(* CODESYS project EAS_SCADA_BATCH.library
   Company: ESCARRE AUTOMATIZACION Y SERVICIOS sl
   Description: 1.1.3
      VAriable ALT fer IN_out
      1.1.2
      Incluir gestion PE
      1.1.1 
      Ajuste comunicacion ADS
      Ajuste tamaño constantes
   Version: 1.1.3
   Placeholder: EAS SCADA BATCH
   Author: EAS
   Title: EAS SCADA BATCH

Project tree, tasks and I/O mapping:
  libraries: Tc2_Standard, * (Beckhoff Automation GmbH); Tc2_System, * (Beckhoff Automation GmbH); Tc3_Module, * (Beckhoff Automation GmbH)
  DUTs/
    PE/
      ELEMENTS/
        data type E_Funcio
        data type PasCicle
        data type T_Compat
        data type T_funcio
        data type T_Sirena
      PE/
        data type PE
        data type PE_COM
      data type ATL
  GVLs/
    global variables Batch
    global variables CONSTANTS
  POUs/
    BATCH/
      function block CarregarFuncionsActivesAlDB [ST]
      function block ComprobarFuncionsPas [ST]
      function block Inic_Func_Actv [ST]
      function block Parar_Func_FiFuncio [ST]
      function block Parar_Func_Incomp [ST]
      function block PararTotesLesFuncions [ST]
      function block Salt [ST]
      function block SaltDePasEnUnCicle [ST]
    GestioPE/
      function block FunBck_v01 [ST]
      function block Func_Activa_v01 [ST]
    program pPE [ST]
  VISUs/
*)

// DUTs/PE/ELEMENTS/E_Funcio
TYPE E_Funcio :
STRUCT

	Cd_Funcio:WORD;
	Actv_Funcio:BOOL;
	ParamFunc:ARRAY [1..Max_ParamFunc] OF WORD;

END_STRUCT
END_TYPE

// DUTs/PE/ELEMENTS/PasCicle
TYPE PasCicle :
STRUCT
	Pas:WORD;
	Funcio:E_Funcio;

END_STRUCT
END_TYPE

// DUTs/PE/ELEMENTS/T_Compat
TYPE T_Compat :
STRUCT

	Funcio1:WORD;  			(*Codi de la primera funcio*)
	Funcio2:WORD;  			(*Codi de la segona funcio*)

END_STRUCT
END_TYPE

// DUTs/PE/ELEMENTS/T_funcio
TYPE T_funcio :
STRUCT

	Cd_funcio:WORD;												(*Codi de la funció*)
	DesFuncio:STRING(16);										(*Descripció de la funció*)
	Background:BOOL;												(*Indicació per si la funció es en backgraund o no*)
	FinFunc:ARRAY [1..max_FinFunc] OF WORD;					(*Funcions que s'han d'acabar al començar aquesta*)

END_STRUCT
END_TYPE

// DUTs/PE/ELEMENTS/T_Sirena
TYPE T_Sirena :
STRUCT
	Actv:BOOL;
	Rearme:BOOL;
END_STRUCT
END_TYPE

// DUTs/PE/PE/PE
TYPE PE :
STRUCT
	///1:manual  2: auto
	wAutoMan: WORD;
	xAuto: BOOL;
	xMan: BOOL;
	///Pas en Automatic, actual o ultim
	wStep: WORD;
	///Función fin de Ciclo
	wFEndCycle: WORD;
	///Tiempo Barcada
	wTBatch: WORD;
	///Tiempo Paso
	wTStep: WORD;
	///Tiempo mantenimiento
	wTMaint: WORD;
	xStartBatch: BOOL;
	xEndBatch: BOOL;
	///array alarmas
	axAlarm: ARRAY[1..Max_Alarmes] OF BOOL;
	///array Sirenas
	axHorn: ARRAY[1..Max_Alarmes] OF BOOL;
	///Pulsador Manual
	xPulMan: BOOL;
	///Pulsador Auto
	xPulAuto: BOOL;
END_STRUCT
END_TYPE

// DUTs/PE/PE/PE_COM
TYPE PE_COM :
STRUCT
	/// -------------------------------------------------------------------- 
	/// InfoBarcada 
	sBatch: STRING(10);
	diNum_Task: DWORD;
	sCdRecipe: STRING(24);
	sDesc_Recipe: STRING(50);
	sCdCycle: STRING(10);
	sDesc_Cycle: STRING(50);
	/// -------------------------------------------------------------------- 
	/// Ordenes PE 
	xToAutomatic: BOOL;
	xToManual: BOOL;
	xToStep: BOOL;
	xRunCycle: BOOL;
	xModifiedCycle: BOOL;
	xStopAlarm: BOOL;
	///Bit Para continuar programa
	xContProg: BOOL;
	///Bit indicacion al iniciar una añadida
	xStartTopping: BOOL;
	///Bit indicacion al finalizar una añadida
	xEndTopping: BOOL;
	///Bit indicacion para resetar los tiempos de la funcion al realizar un salto
	xResetStep: BOOL;
	xReset: BOOL;
	xResetFunc: BOOL;
	///word Per fer un canvi de Pas
	wNewStep: WORD;
	/// Pedir Dosificacion
	axDemandDos: ARRAY[1..max_tanks] OF BOOL;
	/// Numero Dosificacion 
	aiNumDos: ARRAY[1..max_tanks] OF WORD;
	/// OK Peticion Dosificacion
	axOkDemand: ARRAY[1..max_tanks] OF BOOL;
	/// OK  Dosificacion
	axOkDosage: ARRAY[1..max_tanks] OF BOOL;
	/// Tipo Dosificacion 1=Man 2=Auto 3=Mixta
	aiTypeDos: ARRAY[1..max_tanks] OF WORD;
	/// Dosificacion con Producto  Manual *
	axProdMan: ARRAY[1..max_tanks] OF BOOL;
	/// Error Dosificación  *
	axErrorDos: ARRAY[1..max_tanks] OF BOOL;
	/// Volumen dosificat
	aiVolumDos: ARRAY[1..max_tanks] OF DWORD;
	/// Tanque libre 
	axTankFree: ARRAY[1..max_tanks] OF BOOL;
	/// Prioridad
	aiPriority: ARRAY[1..max_tanks] OF WORD;
	/// Solo Disolver
	axOnlyDissol: ARRAY[1..max_tanks] OF BOOL;
END_STRUCT
END_TYPE

// DUTs/PE/ATL
TYPE ATL :
STRUCT
	///------OBLIGATORIO-------------------
	///Sistema PE Com
	PE_COM: PE_COM;
	///Sistema PE 
	PE: PE;
END_STRUCT
END_TYPE

// GVLs/Batch

VAR_GLOBAL RETAIN

(*=======================================	*)
(*					Estat del PE4							*)
(*=======================================	*)

(*Estat de PE4*)
	Func_Comp: ARRAY [1..Max_Compatibles] OF T_Compat;


(*=======================================	*)
(*			Variables de gestió de funcions				*)
(*=======================================	*)

(*Estat de lesFuncions *)
	Est_Func: ARRAY [1..Max_Funcions] OF E_Funcio;  		(*Estat actual de les funcions*)
	Est_F_PE4: ARRAY [1..Max_Funcions] OF E_Funcio;  		(*Estat de les funcions per les comunicacions del PE4*)
	Est_F_PE4_Ant: ARRAY [1..Max_Funcions] OF E_Funcio;  	(*Estat de les funcions per les comunicacions del PE4*)


(* *)
	Config_Func: ARRAY  [1..Max_Funcions] OF t_funcio;		(*Configuració de les funcios *)
	Func_Actives: ARRAY [1..Max_Func_Pas] OF WORD;		(* DB que indica en automaatic les funcions que estan en marcha en automatic*)


(*=======================================	*)
(*			Variables de gestió de cicle					*)
(*=======================================	*)

(*Cicles*)
	Cicle0: ARRAY [1..max_PasCicle] OF PasCicle;  			(*Cicle Actual de treball*)
	CicleRebut: ARRAY [1..max_PasCicle] OF PasCicle;  		(*Cicle Rebut*)


	

(*=======================================	*)
(*			Botons Auto/Man								*)
(*=======================================	*)

	PulsadorManual:BOOL;
	PulsadorAutomatic:BOOL;

(*=======================================	*)
(*			Marcas Internes								*)
(*=======================================	*)

	InicioCiclo:BOOL;


END_VAR


VAR_GLOBAL

(*=======================================	*)
(*			Maquina paralel 								*)
(*=======================================	*)

	TipoParalelo:WORD;
	MaquinaEnParalel:BOOL:=FALSE;
	Master:BOOL;
	Slave:BOOL;
	Pas_M:DWORD;
	Pas_S1:DWORD;
	Pas_S2:DWORD;
	Pas_S3:DWORD;
	Pas_S4:DWORD;
	Tipus_P:DWORD;
	Preparat_C_local:BOOL;
	He_C_local:BOOL;
	Ordre_C:BOOL;
	Ordre_C_Master:BOOL;
	Preparat_C_S1:BOOL;
	Preparat_C_S2:BOOL;
	Preparat_C_S3:BOOL;
	Preparat_C_S4:BOOL;
	He_C_S1:BOOL;
	He_C_S2:BOOL;
	He_C_S3:BOOL;
	He_C_S4:BOOL;
	Fi_C:BOOL;
	Fi_C_master:BOOL;



(*			CONSERVAR  COMPATIBILITAT				*)

	EsperaParalelPerSaltar:BOOL;
	SaltdePas:BOOL;


END_VAR

// GVLs/CONSTANTS

VAR_GLOBAL CONSTANT

(*=======================================	*)
(*			Carregar Constants						*)
(*=======================================	*)
	Max_Funcions:WORD:=128;
	Max_ParamFunc:WORD:=9;
	max_FinFunc:WORD:=5;
	max_PasCicle:WORD:=256;
	Max_Compatibles:WORD:=32;
	Max_Func_Pas:WORD:=12;
	Max_Tanks:WORD:=4;
	Max_Alarmes:WORD:=128;

END_VAR


(*********************************************************************


	Max_ParamFixes:WORD:=150;
	Max_DBFiFuncio: WORD:=640 ;				(* Es calcula com    (Max_Funcions*Max_FinFunc)   *)
	Max_ElementsCicle: WORD:=2816 ;		(* Es calcula com    (Max_PasCicle*(Max_ParamFunc+2))  *)
	Max_DBIncompatibles: WORD:=128;			(* Es calcula com    (Max_Compatibles*2)  *)
	Max_Inputs: WORD:=128;
	Max_Outputs: WORD:=128;
	Max_Analog: WORD:=128;
	Num_Prod_Dos:WORD:=10;         					(* Numero maximo de productos en una dosificación*)
	Max_Prod_Dos:WORD:=128;							(* Productos en una dosificadora*)
	Max_Valv_Dos:WORD:=128;							(* Valvulas en una dosificadora*)
	Max_Alarmes:WORD:=128;



***************************************************************************)

// POUs/BATCH/CarregarFuncionsActivesAlDB
FUNCTION_BLOCK CarregarFuncionsActivesAlDB

(***********************************************************************
Aquest Bloc Carrega les Funcions actives al "DB d'estat de les funcions"
al "DB de funcions actives".   
************************************************************************)

VAR_INPUT
	EstatFuncions: ARRAY [1..max_funcions] OF E_Funcio;
END_VAR

VAR_OUTPUT
	FuncionsActives:ARRAY [1..Max_Func_Pas] OF WORD;
END_VAR

VAR
	Punter:WORD;
	PunterDB:WORD;
	inicialitzaDB: Inic_Func_Actv;
	DB_ple: BOOL;

END_VAR

inicialitzaDB(Func_Actv:= FuncionsActives);
DB_Ple:=FALSE;
punter:=1;
punterDB:=1;
WHILE (punter<=max_funcions)AND NOT(DB_Ple)
	DO
		IF EstatFuncions[punter].Actv_Funcio
			THEN
				FuncionsActives[PunterDB]:=EstatFuncions[punter].Cd_Funcio;
				PunterDB:=PunterDB+1;
				IF punterDB>Max_Func_Pas
					THEN
						DB_ple:=TRUE;
				END_IF
		END_IF
		punter:=punter+1;
END_WHILE

END_FUNCTION_BLOCK

// POUs/BATCH/Inic_Func_Actv
FUNCTION_BLOCK Inic_Func_Actv

(*********************************************************
Reinicia el DB de les funcions actives
***********************************************************)

VAR_IN_OUT
	Func_Actv: ARRAY [1..Max_Func_Pas] OF WORD;		(* DB que indica en automaatic les funcions que estan en marcha en automatic*)
END_VAR

VAR
	Punter: WORD;
END_VAR

Punter:=1;

REPEAT
	Func_Actv[punter]:=0;
	Punter:=Punter+1;
UNTIL
	Punter>Max_Func_Pas
END_REPEAT

END_FUNCTION_BLOCK

// POUs/BATCH/ComprobarFuncionsPas
FUNCTION_BLOCK ComprobarFuncionsPas

(************************************************************
Aquest Bloc Comproba les funcions actves que hi ha en aquest
pas i quan acaben dona l'ordr de canviar de pas.
**************************************************************)

VAR_INPUT
	Estat_F: ARRAY [1..Max_Funcions] OF E_Funcio;
	Tipus_F:ARRAY [1..Max_Funcions] OF T_Funcio;
	FuncionsActives:ARRAY [1..Max_Func_Pas] OF WORD;
END_VAR

VAR_OUTPUT
	AumentaPas:BOOL;
END_VAR

VAR
	Punter: WORD;
	Aumenta: BOOL;
	TempoPAS:TON;

END_VAR

(*Inicialitzar els punters*)
Punter:=1;
Aumenta:=TRUE;

REPEAT
	IF (FuncionsActives[Punter]<>0)AND((Estat_F[FuncionsActives[Punter]].Actv_Funcio=TRUE)AND(Tipus_F[FuncionsActives[Punter]].Background=FALSE))
		THEN
			Aumenta:=FALSE;
	END_IF
	Punter:=Punter+1;
UNTIL
	(Punter>Max_Func_Pas)OR(Aumenta=FALSE)
END_REPEAT

TempoPAS
	(IN:=Aumenta ,
	PT:=t#500ms ,
	Q=>AumentaPas ,
	ET=> );

END_FUNCTION_BLOCK

// POUs/BATCH/Parar_Func_FiFuncio
FUNCTION_BLOCK Parar_Func_FiFuncio

(**************************************************
Para les funcions del "DB de l'estat de funcions" 
depenen de la funcio de la entreda per "fifuncion"
***************************************************)

VAR_INPUT
	Tipus_Funcio:T_funcio;
END_VAR
VAR_OUTPUT
END_VAR
VAR_IN_OUT
	Estat_F: ARRAY [1..Max_Funcions] OF E_Funcio;
END_VAR
VAR
	PunterFiFunc:WORD;
	FuncioIncompat: WORD;
END_VAR

(*..................	Parar les funcions per fin función..................................	*)
PunterFiFunc:=1;
WHILE (PunterFiFunc <= max_FinFunc) DO
	FuncioIncompat :=Tipus_funcio.FinFunc[PunterFiFunc];
	IF FuncioIncompat <>0
		THEN
			Estat_F [FuncioIncompat].Actv_Funcio:=FALSE;
	END_IF
	PunterFiFunc:=PunterFiFunc+1;
END_WHILE

END_FUNCTION_BLOCK

// POUs/BATCH/Parar_Func_Incomp
FUNCTION_BLOCK Parar_Func_Incomp
(************************************************************
L'hi introduim una funció i el el bloc para les funcions del 
"DB estat de les funcions" depenen del 
"DB de compatibilitat"
**************************************************************)
VAR_INPUT
	Funcio:WORD;  (*Funcio que s'ha de parar*)
END_VAR

VAR_OUTPUT
END_VAR

VAR_IN_OUT
	DB_Comp:ARRAY [1..Max_Compatibles] OF T_Compat;
	Estat_F: ARRAY [1..Max_Funcions] OF E_Funcio;
END_VAR

VAR
	PunterEstat:WORD;
	PunterComp:WORD;
END_VAR

(*Mirar si hi ha alguna funció incompatible amb la nova funció*)
PunterEstat:=1;
PunterComp:=1;
REPEAT
	IF DB_Comp[PunterComp].Funcio1=Funcio
		THEN
			PunterEstat:=DB_Comp[PunterComp].Funcio2;
			Estat_F[PunterEstat].Actv_Funcio:=FALSE;
	END_IF
	PunterComp:=PunterComp+1;
UNTIL
	(PunterComp>Max_Compatibles)
END_REPEAT

END_FUNCTION_BLOCK

// POUs/BATCH/PararTotesLesFuncions
FUNCTION_BLOCK PararTotesLesFuncions
(********************************************************
Parar totes les funcions del "DB estat"
*********************************************************)
VAR_IN_OUT
	Estat_F: ARRAY [1..Max_Funcions] OF E_Funcio;
END_VAR

VAR
	Punter: WORD;
END_VAR

(*Inicialitzar els punters*)
Punter:=1;


WHILE (Punter <= Max_Funcions) DO
	IF Estat_F[Punter].Actv_Funcio=TRUE
		THEN
			Estat_F [Punter].Actv_Funcio:=FALSE;
	END_IF
	Punter:=Punter+1;
END_WHILE

END_FUNCTION_BLOCK

// POUs/BATCH/Salt
FUNCTION_BLOCK Salt
(************************************************************
Salta del "Pas inicial" al "Pas Final"  del  "BDCicle"
**************************************************************)
VAR_INPUT
	PasInicial:DWORD;
	PasFinal:DWORD;
END_VAR

VAR_IN_OUT


END_VAR

VAR

	FIFuncio:Parar_Func_FiFuncio;
	Incompatibles:Parar_Func_Incomp;
	PunterCicle:WORD;					(* Aquest valor marca la popsició del db de cicle on estem independent del pas de cicle *)
	T_Func_Act:T_Funcio;				(* Funcio que indica el punterCicle *)

	codi: WORD;

	Est_Func_0: ARRAY [1..Max_Funcions] OF E_Funcio;  		(*Estat de les funcions a cero per reiniciar l'estat*)
END_VAR

(*,,,,,,,,,,,,,,,,,,,,Carregar la posició inicial depenen si es salta desde:
				el pas cero: carerega d'un cicle nou
				un pas en concret: salt sobre el cicle que ja està carregat ,,,,,,,,,,,,,,,,,,,,,  *)

IF PasInicial=0
	THEN
		(*Posar Punter al primer pas*)
		PunterCicle:=1;
		(*Inicialitzar el estat de les funcions*)
		Est_Func:=Est_Func_0;
	ELSE
		(*Buscar Punter Cicle del pas inicial*)
		PunterCicle:=0;
		REPEAT
			PunterCicle := PunterCicle+1;
		UNTIL
			(((Cicle0[PunterCicle].Pas=PasInicial)AND(Cicle0[PunterCicle+1].Pas<>PasInicial)) OR (PunterCicle>=max_PasCicle))
		END_REPEAT
		PunterCicle := PunterCicle+1;      (*02/06/05*)
END_IF

(*,,,,,,,,,,,,,,,,,,,,Bucle de control,,,,,,,,,,,,,,,,,,,,,,,,,,,,,,,,,,,,,,,,,,,,,,,,,,,,,,,,,,,,,	*)

REPEAT
(*.................. Carregar la funció del pas............................................. *)
		codi:=Cicle0[PunterCicle].Funcio.Cd_Funcio;
		IF codi<>0 THEN
		T_Func_Act:=Config_Func[codi];
		END_IF
(*..................	Parar les funcions incompatibles..................................	*)
		Incompatibles(
			Funcio:=T_Func_Act.Cd_funcio ,
			DB_Comp:= Func_Comp ,
			Estat_F:= Est_Func );

(*..................	Activar si es en Background ........................................	*)
		IF T_Func_Act.Background=TRUE
			THEN
				Est_Func[T_Func_Act.Cd_Funcio] := Cicle0[PunterCicle].Funcio ; 	(*Carregar parametres*)
				Est_Func[T_Func_Act.Cd_Funcio].Actv_Funcio:=TRUE;			(*Posar la funció en actiu*)
		END_IF

(*..................	Parar les funcions per fin función..................................	*)
		FiFuncio(
			Tipus_Funcio:=  T_Func_Act ,
			 Estat_F:=Est_Func	 );

(*,,,,,,,,,,,,,,,,,,	Activar funció,,,,,,,,,,,,,,,,,,,,,,,,,,,,,,,,,,,,,,,,,,,,,,,,,,,,,,,,,,,,,,,,,,,	*)
		IF Cicle0[PunterCicle].Pas = PasFinal
			THEN
				Est_Func[T_Func_Act.Cd_Funcio] := Cicle0[PunterCicle].Funcio ;	(*Carregar parametres*)
				Est_Func[T_Func_Act.Cd_Funcio].Actv_Funcio := TRUE;			(*Posar la funció en actiu*)
		END_IF

(*,,,,,,,,,,,,,,,,,,Aumentar el Punter del cicle,,,,,,,,,,,,,,,,,,,,,,,,,,,,,,,,,,,,,,,,,,	*)
		PunterCicle := PunterCicle+1;

UNTIL
	(((Cicle0[PunterCicle].Pas <> PasFinal)AND(Cicle0[PunterCicle-1].Pas = PasFinal))
	OR(PunterCicle>max_PasCicle)
	OR(Cicle0[PunterCicle-1].Funcio.Cd_Funcio=0))
END_REPEAT

END_FUNCTION_BLOCK

// POUs/BATCH/SaltDePasEnUnCicle
FUNCTION_BLOCK SaltDePasEnUnCicle
(************************************************************
Salta del "Pas inicial" al "Pas Final"  del  "BDCicle"
**************************************************************)
VAR_INPUT
	PasInicial:DWORD;
	PasFinal:DWORD;
END_VAR

VAR_IN_OUT


END_VAR

VAR

	FIFuncio:Parar_Func_FiFuncio;
	Incompatibles:Parar_Func_Incomp;
	PunterCicle:WORD;					(* Aquest valor marca la popsició del db de cicle on estem independent del pas de cicle *)
	T_Func_Act:T_Funcio;				(* Funcio que indica el punterCicle *)

	codi: WORD;

	Est_Func_0: ARRAY [1..Max_Funcions] OF E_Funcio;  		(*Estat de les funcions a cero per reiniciar l'estat*)
END_VAR

(*,,,,,,,,,,,,,,,,,,,,Carregar la posició inicial depenen si es salta desde:
				el pas cero: carerega d'un cicle nou
				un pas en concret: salt sobre el cicle que ja està carregat ,,,,,,,,,,,,,,,,,,,,,  *)

IF PasInicial=0
	THEN
		(*Posar Punter al primer pas*)
		PunterCicle:=1;
		(*Inicialitzar el estat de les funcions*)
		Est_Func:=Est_Func_0;
	ELSE
		(*Buscar Punter Cicle del pas inicial*)
		PunterCicle:=0;
		REPEAT
			PunterCicle := PunterCicle+1;
		UNTIL
			(((Cicle0[PunterCicle].Pas=PasInicial)AND(Cicle0[PunterCicle+1].Pas<>PasInicial)) OR (PunterCicle>=max_PasCicle))
		END_REPEAT
		PunterCicle := PunterCicle+1;      (*02/06/05*)
END_IF

(*,,,,,,,,,,,,,,,,,,,,Bucle de control,,,,,,,,,,,,,,,,,,,,,,,,,,,,,,,,,,,,,,,,,,,,,,,,,,,,,,,,,,,,,	*)

REPEAT
(*.................. Carregar la funció del pas............................................. *)
		codi:=Cicle0[PunterCicle].Funcio.Cd_Funcio;
		IF codi<>0 THEN
		T_Func_Act:=Config_Func[codi];
		END_IF
(*..................	Parar les funcions incompatibles..................................	*)
		Incompatibles(
			Funcio:=T_Func_Act.Cd_funcio ,
			DB_Comp:= Func_Comp ,
			Estat_F:= Est_Func );

(*..................	Activar si es en Background ........................................	*)
		IF T_Func_Act.Background=TRUE
			THEN
				Est_Func[T_Func_Act.Cd_Funcio] := Cicle0[PunterCicle].Funcio ; 	(*Carregar parametres*)
				Est_Func[T_Func_Act.Cd_Funcio].Actv_Funcio:=TRUE;			(*Posar la funció en actiu*)
		END_IF

(*..................	Parar les funcions per fin función..................................
		FiFuncio(
			Tipus_Funcio:=  T_Func_Act ,
			 Estat_F:=Est_Func	 );										*)

(*,,,,,,,,,,,,,,,,,,	Activar funció,,,,,,,,,,,,,,,,,,,,,,,,,,,,,,,,,,,,,,,,,,,,,,,,,,,,,,,,,,,,,,,,,,,	*)
		IF Cicle0[PunterCicle].Pas = PasFinal
			THEN
				Est_Func[T_Func_Act.Cd_Funcio] := Cicle0[PunterCicle].Funcio ;	(*Carregar parametres*)
				Est_Func[T_Func_Act.Cd_Funcio].Actv_Funcio := TRUE;			(*Posar la funció en actiu*)
		END_IF

(*,,,,,,,,,,,,,,,,,,Aumentar el Punter del cicle,,,,,,,,,,,,,,,,,,,,,,,,,,,,,,,,,,,,,,,,,,	*)
		PunterCicle := PunterCicle+1;

UNTIL
	(((Cicle0[PunterCicle].Pas <> PasFinal)AND(Cicle0[PunterCicle-1].Pas = PasFinal))
	OR(PunterCicle>max_PasCicle)
	OR(Cicle0[PunterCicle-1].Funcio.Cd_Funcio=0))
END_REPEAT

END_FUNCTION_BLOCK

// POUs/GestioPE/FunBck_v01
FUNCTION_BLOCK FunBck_v01
VAR_INPUT
END_VAR

VAR_OUTPUT
	funcioBck: BOOL;
END_VAR


VAR
	punter: WORD;
END_VAR

punter:=1;
funcioBck:=FALSE;

WHILE ((punter<= Max_Funcions)AND NOT(FuncioBck)) DO
	IF ((Est_func[punter].Actv_funcio)AND NOT(Config_Func[punter].Background))
		THEN
			FuncioBck:=TRUE;
	END_IF
	punter:=punter+1;
END_WHILE

END_FUNCTION_BLOCK

// POUs/GestioPE/Func_Activa_v01
FUNCTION_BLOCK Func_Activa_v01
VAR_INPUT
	EstatFunc:ARRAY [1..Max_Funcions] OF E_Funcio;
END_VAR
VAR_OUTPUT
	FuncionsActives:BOOL;
END_VAR
VAR
	a: WORD;
END_VAR

(*Inicialitza el punter*)
a:=1;
FuncionsActives:=FALSE;
REPEAT
	IF EstatFunc[a].Actv_Funcio=TRUE
		THEN
			FuncionsActives:=TRUE;
	END_IF
	a:=a+1;
UNTIL
(a>Max_Funcions)OR(FuncionsActives=TRUE)
END_REPEAT

END_FUNCTION_BLOCK

// POUs/pPE
PROGRAM pPE
VAR_IN_OUT
	InAtl:ATL;
END_VAR
VAR PERSISTENT
	Anar1: Salt;
	Anar2: Salt;
	Anar3: Salt;
	Anar4: SaltDePasEnUnCicle;
	Anar5: SaltDePasEnUnCicle;
	Parar: PararTotesLesFuncions;
	PararInici: PararTotesLesFuncions;
	ComprobarSalt: ComprobarFuncionsPas;
	SaltarProximPas: BOOL;
	EsperaSalt: TON;
	AcualitzaDB: CarregarFuncionsActivesAlDB;
	AcualitzaDB2: CarregarFuncionsActivesAlDB;
	PunterCicle0: WORD;
	ferSalt: BOOL;
	///ordre de salt
	FerSaltParalel: BOOL;
	EsperaSaltar: TON;
	SaltarPar: BOOL;
	PararTot: PararTotesLesFuncions;
	///=========================================================
	///========  GESTIÓ MANUAL  ================================
	Punt_Func: WORD;
	/// Funcio que indica el punterCicle 
	T_Func_Act: T_Funcio;
	FiFuncio: Parar_Func_FiFuncio;
	Incompatibles: Parar_Func_Incomp;
	a: WORD;
	AcualitzaDB3: CarregarFuncionsActivesAlDB;
	///=========================================================
	fbFUNBCK: FunBck_v01;
	xFunBck: BOOL;
	tFunBck: Ton;
	tCicloOn: ton;
	rsBatch: Rs;
END_VAR
VAR
	run: BOOL;
	inici: Ton;
	xCargadas: BOOL;
	xUltimas: BOOL;
	xBackup: BOOL;
END_VAR


(*==============================================================*)
(*		GESTION REMANENTES PARA CPU CX8190  					*)
(*==============================================================*)

(*==============================================================*)
(*		GESTION PE												*)
(*==============================================================*)
(*,,,,,,,,,,,,,,,,,,,,,,,,,,,,,,,,,,,,,,,,,,,,,Pasar a manual al reiniciar  ,,,,,,,,,,,,,,,,,,,,,,,,,,,,,,,,,,,,,,,,,,,,,,,	*)
inici(IN:= run, PT:=T#5S , Q=> , ET=> );


IF NOT inici.Q THEN
InAtl.PE_COM.xToManual:=TRUE;
InAtl.PE.wAutoMan:=1;
InAtl.PE_COM.xResetFunc:=TRUE;
PararInici(Estat_F:=est_func );
run:=TRUE;
END_IF



(*,,,,,,,,,,,,,,,,,,,,,,,,,,,,,,,,,,,,,,,,,,,,, Orde de Ejecutar Cicle    ,,,,,,,,,,,,,,,,,,,,,,,,,,,,,,,,,,,,,,,,,,,,,,,,,,,,	*)

IF InAtl.PE_COM.xRunCycle
	THEN
		Cicle0:=CicleRebut;
		InAtl.PE.wStep :=0;
		InAtl.PE.wAutoMan:=2;
		Anar2(
			PasInicial:= 0 ,
			 PasFinal:= InAtl.PE.wStep );
		InAtl.PE_COM.xRunCycle:= FALSE;
END_IF

(*,,,,,,,,,,,,,,,,,,,,,,,,,,,,,,,,,,,,,,,,,,,,,Orde de Cicle Modificat ,,,,,,,,,,,,,,,,,,,,,,,,,,,,,,,,,,,,,,,,,,,,,,,,	*)
IF InAtl.PE_COM.xModifiedCycle
	THEN
		Cicle0:=CicleRebut;
		InAtl.PE_COM.xModifiedCycle:=FALSE;
END_IF

(*,,,,,,,,,,,,,,,,,,,,,,,,,,,,,,,,,,,,,,,,,,,,,Orde de Reset ,,,,,,,,,,,,,,,,,,,,,,,,,,,,,,,,,,,,,,,,,,,,,,,,,,,,,,,,,,,,,,,,	*)
IF InAtl.PE_COM.xReset
	THEN
		PararTot(Estat_F:=Est_F_PE4 );
		InAtl.PE.wStep :=0;
		InAtl.PE_COM.xToManual:=TRUE;
		InAtl.PE_COM.xReset:=FALSE;
END_IF
(*,,,,,,,,,,,,,,,,,,,,,,,,,,,,,,,,,,,,,,,,,,,,,Orde de Reset ,,,,,,,,,,,,,,,,,,,,,,,,,,,,,,,,,,,,,,,,,,,,,,,,,,,,,,,,,,,,,,,,	*)
IF InAtl.PE_COM.xResetFunc
	THEN
		PararTot(Estat_F:=Est_F_PE4 );
		InAtl.PE_COM.xResetFunc :=FALSE;
END_IF


(*=============================================================*)
(*=============================================================*)

(*Control si el sistema treballa en MANUAL / AUTOMATIC *)

(*,,,,,,,,,,,,,,,,,,,,,,,,,,,,,,,,,,,,,,,, Canvis d'estat AUTO/MAN ,,,,,,,,,,,,,,,,,,,,,,,,,,,,,,,,,,,,,,,,,,,,,,,,,	*)
(*  Automàtic   *)
IF ((InAtl.PE.xPulAuto)(*OR Com_PE.RetardArranc*) OR (InAtl.PE_COM.xToAutomatic) OR (InAtl.PE.wAutoMan>2))AND(cicle0[1].Pas<>0)
	THEN
		(* Pasar de Manual a Automatic*)
		IF InAtl.PE.wAutoMan<=1
			THEN
				Parar(Estat_F:=Est_Func);
				IF InAtl.PE.wStep=0
					THEN
						InAtl.PE.wStep:=1;
				END_IF
				Anar3(
					PasInicial:= 0 ,
		 			PasFinal:= InAtl.PE.wStep );
		END_IF
		InAtl.PE.wAutoMan:=2;
		AcualitzaDB
			(EstatFuncions:= Est_Func  ,
			FuncionsActives=>Func_Actives );
END_IF;
		InAtl.PE_COM.xToAutomatic:=FALSE;

(*  Manual   *)
IF (InAtl.PE.xPulMan) OR (InAtl.PE_COM.xToManual) OR (InAtl.PE.wAutoMan<1)
	THEN
		(* Pasar d'automatic a manual *)
		IF InAtl.PE.wAutoMan>=2
			THEN
				Parar(Estat_F:=Est_Func);
		END_IF
		InAtl.PE.wAutoMan:=1;
		InAtl.PE_COM.xToManual:=FALSE;
END_IF;


(*=============================================================*)
(* + + + + + + + +  +  + + + + + + + + + + + + + + + + + + + + + + + + + + + + + + + + + *)

(*,,,,,,,,,,,,,,,,,,,,,,,,,,,,,,,,,,,,,,,,,, Gestio Manual,,,,,,,,,,,,,,,,,,,,,,,,,,,,,,,,,,,,,,,,,,,,,,,,,,,,,,,,,,,,,,,,,,,,,	*)

IF InAtl.PE.wAutoMan=1
	THEN
(*_____________________________________________________________________________________________________________*)
		Punt_Func:=1;
		REPEAT
			IF (Est_Func[Punt_Func].Actv_Funcio)=(Est_F_PE4[Punt_Func].Actv_Funcio)
			THEN
				(*Igualar valors de les funcions*)
				Est_Func[Punt_Func]:=Est_F_PE4[Punt_Func];
				(*Aumentar el punter*)
				Punt_Func:=Punt_Func+1;
			ELSE
				T_Func_Act:=Config_Func[Punt_Func];
				IF Est_Func[Punt_Func].Actv_Funcio=TRUE
				THEN
					(* Parar la funcio al PLC per fi funcio manual al PE4  *)
					Est_Func[Punt_Func].Actv_Funcio:=FALSE;
				ELSE
					IF (Est_F_PE4[Punt_Func].Actv_Funcio=TRUE)AND(Est_F_PE4_Ant[Punt_Func].Actv_Funcio=TRUE)
					THEN
						(*Parar la funcio al PE4 per que s'ha acabat*)
							Est_F_Pe4[Punt_Func].Actv_Funcio:=FALSE;
					ELSE
						(*=====Activar la funció====*)
						(*Mirar si hi ha alguna funció incompatible amb la nova funció*)
						Incompatibles(
							Funcio:= T_Func_Act.Cd_funcio ,
							DB_Comp:= Func_Comp,
							Estat_F:=Est_Func );
		
						(*Mirar si la funcio nova ha d'acabar alguna funció per Fin Funcion*)
						FiFuncio(
							Tipus_Funcio:= T_Func_Act ,
							Estat_F:= Est_func);
						(*Activar la funció*)
						Est_Func[Punt_Func]:= Est_F_PE4[Punt_Func];
					END_IF
				END_IF
			END_IF
		UNTIL
		Punt_Func>Max_Funcions
		END_REPEAT
		AcualitzaDB3
			(EstatFuncions:= Est_Func  ,
			FuncionsActives=>Func_Actives );
		
		Est_F_PE4_Ant:=Est_F_PE4;
(*_____________________________________________________________________________________________________________*)
		SaltarProximPas:=FALSE;
END_IF


(*=============================================================*)
(* + + + + + + + +  +  + + + + + + + + + + + + + + + + + + + + + + + + + + + + + + + + + *)
(*,,,,,,,,,,,,,,,,,,,,,,,,,,,,,,,,,,,,, Gestio En Autiomatic,,,,,,,,,,,,,,,,,,,,,,,,,,,,,,,,,,,,,,,,,,,,,,,,,,,,,,,,,,,,,	*)


IF InAtl.PE.wAutoMan=2
	THEN
		(*__________________Comprobar si cal pasar la seguent PAS_______________________________________________*)
		ComprobarSalt(
			Estat_F:= Est_Func,
			Tipus_F:=Config_Func ,
			FuncionsActives:= Func_Actives,
			AumentaPas=> SaltarProximPas );

		(*__________________Buscar Punter Cicle del pas inicial___________________________________________________*)

	PunterCicle0:=0;
		REPEAT
			PunterCicle0 := PunterCicle0+1;
		UNTIL
			(((Cicle0[PunterCicle0].Pas=InAtl.PE.wStep)AND(Cicle0[PunterCicle0+1].Pas<>InAtl.PE.wStep)) OR (PunterCicle0>=max_PasCicle))
		END_REPEAT

		(*__________________Fer Canvi de pas _______________________________________________________________*)
		IF SaltarProximPas AND NOT he_C_local
			THEN
				IF NOT(MaquinaEnParalel)
				THEN
				(* ·······················Maquina Single o Paralel desacoplada ··············································································································· *)
				Anar4(
					PasInicial:= InAtl.PE.wStep,
		 			PasFinal:= (InAtl.PE.wStep + 1) );
				InAtl.PE.wStep:=InAtl.PE.wStep + 1;
				SaltarProximPas:=FALSE;
				AcualitzaDB(
					EstatFuncions:= Est_Func  ,
					FuncionsActives=>Func_Actives );
				ELSE
				(* ·······················Maquina  En Paralel Acoplada ··························································································································· *)
				(*---------------------------------------------------------------------------------------------------------------------------------------------------------*)
				(*........................Indicar que la maquina local està preparada per pasar de pas..........................:........................................*)
				Preparat_C_local:=TRUE;
				(*........................Ordre de canvi ::::..........::::::::::.........::::::::::.........::::::::::.........::::::::::.........::::::::::.........::::::::::.........::::::::::.........:::::.*)
				(*........................Maquina Master: Actv ordre de canvi de pas.::::::::::.........::::::::::.........::::::::::.........::::::::::.........::::::::::.........:::::.*)
				(* 10/06/2011   preparat per diferents tipus de paralel   *)
				IF tipoparalelo<=2 THEN
					Ordre_C:= Master AND Preparat_C_local AND Preparat_C_S1;
				END_IF
				IF tipoparalelo=3 THEN
					Ordre_C:= Master AND Preparat_C_local AND Preparat_C_S1 AND Preparat_C_S2;
				END_IF
				IF tipoparalelo=4 THEN
					Ordre_C:= Master AND Preparat_C_local AND Preparat_C_S1 AND Preparat_C_S2 AND Preparat_C_S3;
				END_IF
				IF tipoparalelo>=5 THEN
					Ordre_C:= Master AND Preparat_C_local AND Preparat_C_S1 AND Preparat_C_S2 AND Preparat_C_S3 AND Preparat_C_S4;
				END_IF

				(*........................Activar el canvi procedent del master ..........::::::::::.........::::::::::.........::::::::::.........::::::::::.........::::::::::.........:::::.*)
				FerSaltParalel:=Ordre_C_Master AND NOT He_C_local;
				(*"""""""""""""Ordre de saltar,,,,,,,,,,,,,,,,,,,,,,,,,,,,,,,,,,,,,,,,,,,,,,,,,,,,,,,,,,,,,,,,,,,,,,,,,,,,,,,,,,,,,,,,,,,,,,,,,,,,,,,,,,,,,,,,,,,,,,,,,,,,,,,,,,,,,,,,,,,,,,,,,,,,,,,,,,,,,,*)
				IF  SaltarPar THEN
					Anar5(
						PasInicial:= InAtl.PE.wStep,
		 				PasFinal:= (InAtl.PE.wStep+1) );
					InAtl.PE.wStep:=InAtl.PE.wStep+1;
					SaltarProximPas:=FALSE;
					AcualitzaDB2(
						EstatFuncions:= Est_Func  ,
						FuncionsActives=>Func_Actives );
				(*........................Marca local  que ja s'ha fet el salt ::::..........::::::::::.........::::::::::.........::::::::::.........::::::::::.........::::::::::.........:::::.*)
					He_C_local:=TRUE;                            (* Marca de salt fet *)
				END_IF
			END_IF
		END_IF
		Est_F_PE4_Ant:=Est_F_PE4;
		Est_F_PE4:=Est_Func;
END_IF

(*Espera per asegurar que no es fa més de un salt de cop*)
EsperaSaltar(IN:= FerSaltParalel, PT:=t#1s , Q=>SaltarPar );

(*........................Maquina Master: Comprobar que tots han fet el canvi:::::::::.........::::::::::.........::::::::::.........::::::::::.........:::::.*)
(* 10/06/2011   preparat per diferents tipus de paralel   *)
IF tipoparalelo<=2 THEN
	Fi_C:= ( Master AND He_C_local AND He_C_S1 )OR( master AND Fi_C AND Preparat_C_S1);
END_IF
IF tipoparalelo=3 THEN
	Fi_C:= ( Master AND He_C_local AND He_C_S1 AND He_C_S2 )OR( master AND Fi_C AND (Preparat_C_S1 OR Preparat_C_S2));
END_IF
IF tipoparalelo=4 THEN
	Fi_C:= ( Master AND He_C_local AND He_C_S1 AND He_C_S2 AND He_C_S3 )OR( master AND Fi_C AND (Preparat_C_S1 OR Preparat_C_S2 OR Preparat_C_S3));
END_IF
IF tipoparalelo>=5 THEN
	Fi_C:= ( Master AND He_C_local AND He_C_S1 AND He_C_S2 AND He_C_S3 AND He_C_S4 )OR( master AND Fi_C AND (Preparat_C_S1 OR Preparat_C_S2 OR Preparat_C_S3 OR Preparat_C_S4));
END_IF



(*........................Fer Reset dels valors per fi de canvi de pas::::::::::::::::::::::::::.........::::::::::.........::::::::::.........::::::::::.........:::::.*)
IF Fi_C_Master OR InAtl.PE.wAutoMan<=1 OR NOT(MaquinaEnParalel) THEN
	Preparat_C_local:=FALSE;
	Preparat_C_S1:=FALSE;
	Preparat_C_S2:=FALSE;
	Preparat_C_S3:=FALSE;
	Preparat_C_S4:=FALSE;
	He_C_local:=FALSE;
	He_C_S1:=FALSE;
	He_C_S2:=FALSE;
	He_C_S3:=FALSE;
	He_C_S4:=FALSE;
	Ordre_C:=FALSE;
	Ordre_C_Master:=FALSE;
	FerSaltParalel:=FALSE;
	SaltarPar:=FALSE;
END_IF

(* Reset valors paralel en cas de manual*)
IF InAtl.PE.wAutoMan=1
	THEN
	FerSaltParalel:=FALSE;
END_IF

(*,,,,,,,,,,,,,,,,,,,,,,,,,,,,,,,,,,,,,,,,,,,,,Orde de Salt de pas ,,,,,,,,,,,,,,,,,,,,,,,,,,,,,,,,,,,,,,,,,,,,,,,,,,,,,,,,	*)
EsperaSalt(IN:= InAtl.PE_COM.xToStep, PT:=T#2S , Q=>ferSalt , ET=> );
IF ferSalt 
	THEN
		Parar(Estat_F:= Est_Func );
		Anar1(
			PasInicial:= 0 ,
			PasFinal:= InAtl.PE_COM.wNewStep );
		InAtl.PE.wStep:=InAtl.PE_COM.wNewStep;
		InAtl.PE_COM.xResetStep:=TRUE;
		InAtl.PE_COM.xToStep:= FALSE;
END_IF
AcualitzaDB(
	EstatFuncions:= Est_Func  ,
	FuncionsActives=>Func_Actives );


(*=====================================================================================================================================*)
(* INDICACIONS AUTO MAN*)

InAtl.PE.xMan := InAtl.PE.wAutoMan= 1  ;
InAtl.PE.xAuto := InAtl.PE.wAutoMan= 2  ;

(*=====================================================================================================================================*)
(*CALCULO DURACION PASO*)
fbFUNBCK(funcioBck=>xFunBck );
tFunBck(IN:=xFunBck , PT:=T#10D );
InAtl.PE.wTStep := REAL_TO_WORD((TIME_TO_REAL(tFunBck.ET))/1000.0); (*expresado en segundos*)
(*=====================================================================================================================================*)
(*CALCULO DURACION BARCADA*)
rsBatch(SET:=InAtl.PE.xStartBatch , RESET1:=InAtl.PE.xEndBatch );
tCicloOn(IN:= rsBatch.Q1, PT:=T#10D );
InAtl.PE.wTBatch:= REAL_TO_WORD((TIME_TO_REAL(tCicloOn.ET))/60000.0);(*expresado en minutos*)
(*=====================================================================================================================================*)

END_PROGRAM
